// TIA Portal V17 export
// export: Created 2024-09-15T12:30:38.1838598Z, ExportSetting WithDefaults, DisplayName Totally Integrated Automation Portal, DisplayVersion V17, DisplayName TIA Portal Openness, DisplayVersion V17, DisplayName TIA Portal Version Control Interface, DisplayVersion V17, DisplayName STEP 7 Professional, DisplayVersion V17, DisplayName STEP 7 Safety, DisplayVersion V17, DisplayName WinCC Professional, DisplayVersion V17
TYPE "typ_Tracking"
// stored: IsFailsafeCompliant false
   STRUCT
      track_puck : String;
   END_STRUCT;
END_TYPE
